(* POU GENERAL/FB_CALC_TOOLTENSION_FORCE_NEW, ST *)
FUNCTION_BLOCK FB_CALC_TOOLTENSION_FORCE_NEW
VAR_INPUT
	rForcePistonIn:REAL;	(* in Newton *)
	rPistonDiameterD1:REAL;	(* in mm *)
	rPistonDiameterD2:REAL;	(* in mm *)
	rMaxAirpressure:REAL;		(* in bar *)
	rFactorForce:REAL;
END_VAR
VAR_OUTPUT
	iAnalogOutput:INT;		(* range 0 - 32767 *)
	rSetMaxForce:REAL;		(* in Newton *)
	rForcePistonOut:REAL;	(* in Newton *)
END_VAR
VAR
	rMaxForce: REAL;
	rAreaOutside: REAL;
	rAreaInside: REAL;
	rArea: REAL;
	rTmpMaxAirpressure: REAL;
	rTmpAnalogOut:REAL;
END_VAR
(****************************************************************************************************************************************************)
(*****       This Functionblock calculate the effective value for the servo ventil for the ToolTension which the settled force         *****)
(****************************************************************************************************************************************************)
	rAreaOutside:=((rPistonDiameterD1/2)*(rPistonDiameterD1/2))*PI;
	rAreaInside:=((rPistonDiameterD2/2)*(rPistonDiameterD2/2))*PI;
	rArea:=ABS(rAreaOutside - rAreaInside);
	rArea:=rArea / 1000000.0;	(* Umwandeln von mm^2 in m^2 *)
	rTmpMaxAirpressure:=rMaxAirpressure * 100000.0;	(* convert from bar to pascal *)
	rMaxForce:=rArea * rTmpMaxAirpressure * rFactorForce;
	rSetMaxForce:=rMaxForce;

	IF(rMaxForce = 0) THEN rMaxForce:=0.01; END_IF;	(* check divide by zero *)
	IF(rMaxForce <> 0.0) THEN
		rTmpAnalogOut:=(rForcePistonIn/rMaxForce)*32767;	(* 32767 = 10V *)
		IF (rTmpAnalogOut > 32767) THEN
			iAnalogOutput:=32767;
		ELSE
			iAnalogOutput:=REAL_TO_INT(rTmpAnalogOut);
		END_IF;
		rForcePistonOut:=rForcePistonIn;
	ELSE
		iAnalogOutput:=0;
		rForcePistonOut:=0;
	END_IF;
END_FUNCTION_BLOCK

(* POU FB_HARDWARE/FBHW_CYL_STANDARD, ST *)
FUNCTION_BLOCK FBHW_CYL_STANDARD
VAR_INPUT
	xCtrlePosOn:BOOL;
	xCtrlePosOff:BOOL;
END_VAR
VAR_OUTPUT
	xCylinder:BOOL;
END_VAR
VAR_IN_OUT
	T_Cylinder:ST_CYLINDER;
END_VAR
VAR
(* variable *)
	xConfirmResetFB:BOOL:=FALSE;
	iStep:INT;
(* timer *)
	TimerOn:TON;
	TimerOff:TON;
	TimerPreOn:TON;
	TimerPreOff:TON;
	TimerOut:TON;
	TimerActiv: TON;
(* trigger *)
	RisingEdgeActiv:R_TRIG;
	FallingEdgeActiv:F_TRIG;
	RisingEdgeReset:R_TRIG;
	RisingEdgeExecute:R_TRIG;
	TimerAfterSensor: TON;
END_VAR
(* if function bloc set activ then Analog state will be transfered *)
	RisingEdgeActiv(CLK:=T_Cylinder.T_CtrleCyl.xFBActiv);
	FallingEdgeActiv(CLK:=T_Cylinder.T_CtrleCyl.xFBActiv);
	IF RisingEdgeActiv.Q OR FallingEdgeActiv.Q THEN
	(* set Analog Out = In on the rising edge from the activ signal *)
		xCylinder:=NOT(T_Cylinder.T_Config.xActivState);
		T_Cylinder.T_CtrleCyl.T_Standard.xActivOn:= FALSE;
	END_IF

(* if bloc disable if activ signal is inactiv *)
	IF T_Cylinder.T_CtrleCyl.xFBActiv THEN
	(* copy control position state *)
		T_Cylinder.T_CtrleCyl.xStatePosOn:=xCtrlePosOn;
		T_Cylinder.T_CtrleCyl.xStatePosOff:=xCtrlePosOff;
	ELSE
	(* exit FB *)
		T_Cylinder.T_CtrleCyl.xStatePosOn:=xCtrlePosOn;
		T_Cylinder.T_CtrleCyl.xStatePosOff:=xCtrlePosOff;
		RETURN;
	END_IF

(* wait for reseting *)
	RisingEdgeReset(CLK:=T_Cylinder.T_CtrleCyl.xReset);
	IF RisingEdgeReset.Q THEN
		(* Init. timer *)
		TimerOn(IN:=TRUE,PT:=T#1ms);
		TimerOff(IN:=TRUE,PT:=T#1ms);
		TimerPreOn(IN:=TRUE,PT:=T#1ms);
		TimerPreOff(IN:=TRUE,PT:=T#1ms);
		TimerOut(IN:=TRUE,PT:=T#1ms);
	(* Init. variable *)
		iStep:=0;
	(* Init. structure *)
		T_Cylinder.T_CtrleCyl.iFunction:=0;
		T_Cylinder.T_CtrleCyl.T_Standard.xActivOn:=FALSE;
		xCylinder:=NOT(T_Cylinder.T_Config.xActivState);
		T_Cylinder.T_CtrleCyl.xDone:=FALSE;
		T_Cylinder.T_CtrleCyl.xErr:=FALSE;
		T_Cylinder.T_CtrleCyl.udiErrorID:=16#0;
	(* confirm reset *)
		xConfirmResetFB:=TRUE;
	(* exit function *)
		RETURN;
	ELSE
		IF xConfirmResetFB THEN
		(* confirm reset FB *)
			T_Cylinder.T_CtrleCyl.xDone:=TRUE;
			T_Cylinder.T_CtrleCyl.xErr:=FALSE;
			T_Cylinder.T_CtrleCyl.udiErrorID:=16#0;
			(* reset variable *)
			xConfirmResetFB:=FALSE;
		END_IF
	END_IF

(* if bloc disable if activ signal is inactiv *)
	IF NOT(T_Cylinder.T_CtrleCyl.xFBActiv) THEN
		RETURN;
	END_IF

(* wait for execute *)
	RisingEdgeExecute(CLK:=T_Cylinder.T_CtrleCyl.xExecute);
	IF RisingEdgeExecute.Q THEN
		IF NOT(T_Cylinder.T_CtrleCyl.xDone) AND NOT(T_Cylinder.T_CtrleCyl.xErr) THEN
		(* can execute function if both signal are disable *)
			RETURN;
		END_IF
		CASE T_Cylinder.T_CtrleCyl.iFunction OF
		(* disable *)
		1:	iStep:=11;
		(* Activ without sensor position ctrle *)
		2:	iStep:=1;
		(* inverse cylinder state *)
		51:	iStep:=51;
		ELSE
			(* function not implemented *)
			iStep:=0;
			T_Cylinder.T_CtrleCyl.xDone:=FALSE;
			T_Cylinder.T_CtrleCyl.xErr:=TRUE;
			T_Cylinder.T_CtrleCyl.udiErrorID:=16#F000;
			(* exit FB *)
			RETURN;
		END_CASE
		(* Init. variable *)
		T_Cylinder.T_CtrleCyl.xDone:=FALSE;
		T_Cylinder.T_CtrleCyl.xErr:=FALSE;
		T_Cylinder.T_CtrleCyl.udiErrorID:=16#0;
		(* exit FB *)
		RETURN;
	END_IF

(* Timer activ *)
	TimerOn(IN:=TRUE,PT:=T_Cylinder.T_Config.tDelayOn);
	TimerOff(IN:=TRUE,PT:=T_Cylinder.T_Config.tDelayOff);
	TimerPreOn(IN:=TRUE,PT:=T_Cylinder.T_Config.tDelayPreOn);
	TimerPreOff(IN:=TRUE,PT:=T_Cylinder.T_Config.tDelayPreOff);
	TimerOut(IN:=TRUE,PT:=T_Cylinder.T_Config.tTimeOut);
	TimerActiv(IN:=TRUE,PT:=T_Cylinder.T_CtrleCyl.T_Standard.tDelayActiv);
	TimerAfterSensor(IN:=TRUE,PT:=T_Cylinder.T_CtrleCyl.T_Standard.tDelayAfterSensor);
(* waiting for activ *)
	CASE iStep OF
	(* process timer On *)
	1:	IF (T_Cylinder.T_Config.tDelayPreOn = T#0s) THEN
			TimerOn(IN:=FALSE);
			xCylinder:=T_Cylinder.T_Config.xActivState;
			T_Cylinder.T_CtrleCyl.T_Standard.xActivOn:=TRUE;
			iStep:=2;
		ELSE
			TimerPreOn(IN:=FALSE);
			iStep:=4;
		END_IF;
	(* wait for timer On *)
	2:	IF TimerOn.Q THEN
			iStep:=3;
			TimerOut(IN:=FALSE);
		END_IF
	(* control position activ *)
	3:	IF T_Cylinder.T_Config.xCtrlePosOn THEN
		(* position ctrle activ *)
			IF TimerOut.Q THEN
			(* timerout done, activ error cylinder has not activ position reached *)
				iStep:=999;
			ELSE
				IF xCtrlePosOn THEN
				(* Activ position reached, activ confirmation *)
					iStep:=80;
				END_IF
			END_IF
		ELSE
		(* no position ctrle, activ confirm *)
			iStep:=90;
		END_IF
	(* wait for timer Pre On *)
	4:	IF TimerPreOn.Q THEN
			T_Cylinder.T_Config.tDelayPreOn:=T#0s;
			iStep:=1;
		END_IF
	(* process timer Off *)
	11:	IF (T_Cylinder.T_Config.tDelayPreOff = T#0s) THEN
			TimerOff(IN:=FALSE);
			xCylinder:=NOT(T_Cylinder.T_Config.xActivState);
			T_Cylinder.T_CtrleCyl.T_Standard.xActivOn:=FALSE;
			iStep:=12;
		ELSE
			TimerPreOff(IN:=FALSE);
			iStep:=14;
		END_IF;
	(* wait for timer Off *)
	12:	IF TimerOff.Q THEN
			iStep:=13;
			TimerOut(IN:=FALSE);
		END_IF
	(* control position inactiv *)
	13:	IF T_Cylinder.T_Config.xCtrlePosOff THEN
		(* control position activ *)
			IF TimerOut.Q THEN
			(* timerout done, activ error 'cylinder has not inactiv position reached' *)
				iStep:=998;
			ELSE
				IF xCtrlePosOff THEN
				(* inactiv position reached, activ confirmation *)
					iStep:=85;
				END_IF
			END_IF
		ELSE
		(* no control position activ, activ confirmation *)
			iStep:=99;
		END_IF
	(* wait for timer Pre Off *)
	14:	IF TimerPreOff.Q THEN
			T_Cylinder.T_Config.tDelayPreOff:=T#0s;
			iStep:=11;
		END_IF
	(* inverse cylinder state *)
	51:	xCylinder:=NOT(xCylinder);
		T_Cylinder.T_CtrleCyl.T_Standard.xActivOn:=NOT(T_Cylinder.T_CtrleCyl.T_Standard.xActivOn);
		iStep:=99;
	80:	IF (T_Cylinder.T_CtrleCyl.T_Standard.tDelayAfterSensor <> T#0s) THEN
			TimerAfterSensor(IN:=FALSE);
			iStep:=81;
		ELSE
			iStep:=90;
		END_IF;
	(* wait for time after sensor *)
	81:	IF TimerAfterSensor.Q THEN
			iStep:=90;
		END_IF
	85:	IF (T_Cylinder.T_CtrleCyl.T_Standard.tDelayAfterSensor <> T#0s) THEN
			TimerAfterSensor(IN:=FALSE);
			iStep:=86;
		ELSE
			iStep:=99;
		END_IF;
	(* wait for time after sensor *)
	86:	IF TimerAfterSensor.Q THEN
			iStep:=99;
		END_IF
	(* test if delay activ *)
	90:	IF T_Cylinder.T_CtrleCyl.T_Standard.tDelayActiv <> T#0s THEN
			TimerActiv(IN:=FALSE);
			iStep:=98;
		ELSE
			iStep:=99;
		END_IF
	(* wait for time delay activ *)
	98:	IF TimerActiv.Q THEN
		(* activ time is over, set variable off *)
			xCylinder:=NOT(T_Cylinder.T_Config.xActivState);
			T_Cylinder.T_CtrleCyl.T_Standard.xActivOn:=FALSE;
			iStep:=99;
		END_IF
	(* process end *)
	99:	T_Cylinder.T_CtrleCyl.xDone:=TRUE;
		T_Cylinder.T_CtrleCyl.xErr:=FALSE;
		T_Cylinder.T_CtrleCyl.udiErrorID:=16#0;
	(* error, cylinder not in inactiv position *)
	998:	T_Cylinder.T_CtrleCyl.xDone:=FALSE;
		T_Cylinder.T_CtrleCyl.xErr:=TRUE;
		T_Cylinder.T_CtrleCyl.udiErrorID:=16#F202;
	(* error, cylinder not in activ position *)
	999:	T_Cylinder.T_CtrleCyl.xDone:=FALSE;
		T_Cylinder.T_CtrleCyl.xErr:=TRUE;
		T_Cylinder.T_CtrleCyl.udiErrorID:=16#F201;
	END_CASE
END_FUNCTION_BLOCK

(* POU PRG_TWINSAFE, FBD *)
PROGRAM PRG_TWINSAFE
VAR
	TwinSAFEinputKlemme1: TwinSAFE_input;
	TwinSAFEinputKlemme2: TwinSAFE_input;
	TwinSAFEinputKlemme3: TwinSAFE_input;
END_VAR
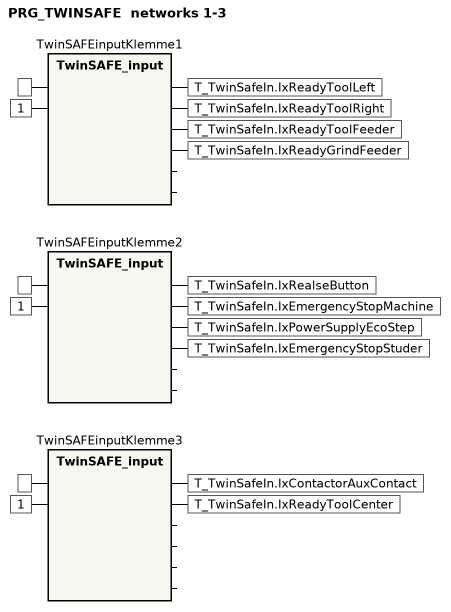
_FBD_ (* Function Block Diagram *)
NETWORK 1 (* Read of the TwinSAFE inputs *)
	TwinSAFEinputKlemme1:TwinSAFE_input(, 1, out 2 => T_TwinSafeIn.IxReadyToolRight, out 3 => T_TwinSafeIn.IxReadyToolFeeder, out 4 => T_TwinSafeIn.IxReadyGrindFeeder) => T_TwinSafeIn.IxReadyToolLeft
NETWORK 2 (* Read of the TwinSAFE inputs *)
	TwinSAFEinputKlemme2:TwinSAFE_input(, 1, out 2 => T_TwinSafeIn.IxEmergencyStopMachine, out 3 => T_TwinSafeIn.IxPowerSupplyEcoStep, out 4 => T_TwinSafeIn.IxEmergencyStopStuder) => T_TwinSafeIn.IxRealseButton
NETWORK 3 (* Read of the TwinSAFE inputs *)
	TwinSAFEinputKlemme3:TwinSAFE_input(, 1, out 2 => T_TwinSafeIn.IxReadyToolCenter) => T_TwinSafeIn.IxContactorAuxContact
_END_FBD_
END_PROGRAM

(* POU PRG_USB_IO_PANEL, ST *)
PROGRAM PRG_USB_IO_PANEL
VAR
(* Panel tastatur *)
	(* function bloc *)
	fbCtrlePanel_IO:FBHW_PANEL_IO;
	(* IO connection *)

	IarxCtrlePanelButton AT %I* : ARRAY[1..10] OF BOOL;
	QarxCtrlePanelLed AT %Q* : ARRAY[1..10] OF BOOL;
END_VAR
(****************************************************************************************************************************************************)
(***********                This Programm Unit make the connection for read and set the ControlPanel Led and Button               ************)
(****************************************************************************************************************************************************)
(* Call FB *)
	fbCtrlePanel_IO(	arxButton:=IarxCtrlePanelButton,
					T_CtrlePanel:=T_CtrlePanel,
					arxLed=>QarxCtrlePanelLed);
END_PROGRAM

(* POU FB_HARDWARE/FBHW_PANEL_IO, ST *)
FUNCTION_BLOCK FBHW_PANEL_IO
VAR_INPUT
	arxButton:ARRAY[1..10] OF BOOL;
END_VAR
VAR_OUTPUT
	arxLed:ARRAY[1..10] OF BOOL;
END_VAR
VAR_IN_OUT
	T_CtrlePanel:ST_CTRLEPANEL;
END_VAR
VAR
(* variable *)
	xConfirmResetFB:BOOL;
	xConfirmFct:BOOL;
	i: INT;
	si: SINT;
(* trigger *)
	RisingEdgeExecute:R_TRIG;
	RisingEdgeReset:R_TRIG;
END_VAR
(****************************************************************************************************************************************************)
(***********                                            This Functionblock is for manage the IO's of the ControlPanel                                             ************)
(****************************************************************************************************************************************************)
(* reset function bloc *)
	RisingEdgeReset(CLK:=T_CtrlePanel.xReset);
	IF RisingEdgeReset.Q THEN
	(* reset output *)
		FOR i := 1 TO 10 DO
			arxLed[i]:=FALSE;
		END_FOR
	(* init. structure *)
		T_CtrlePanel.iFunction:=0;
		T_CtrlePanel.xDone:=FALSE;
		T_CtrlePanel.xErr:=FALSE;
		T_CtrlePanel.udiErrorID:=0;
		T_CtrlePanel.udiButton:=0;
		T_CtrlePanel.udiLED:=0;
	(* confirm reset *)
		xConfirmResetFB:=TRUE;
	(* exit fb *)
		RETURN;
	ELSE
		IF xConfirmResetFB THEN
		(* confirm reset FB *)
			T_CtrlePanel.xDone:=TRUE;
			T_CtrlePanel.xErr:=FALSE;
			T_CtrlePanel.udiErrorID:=0;
			(* Init. variable *)
			xConfirmResetFB:=FALSE;
		END_IF
	END_IF

(* Switch on/off the Led from the control panel *)
	RisingEdgeExecute(CLK:=T_CtrlePanel.xExecute);
	IF RisingEdgeExecute.Q THEN
		CASE T_CtrlePanel.iFunction OF
		(* switch off a specific LED off *)
		-10..-1:	IF arxLed[ABS(T_CtrlePanel.iFunction)] THEN
					arxLed[ABS(T_CtrlePanel.iFunction)]:=FALSE;
					T_CtrlePanel.udiLED:=T_CtrlePanel.udiLED - MUX(ABS(T_CtrlePanel.iFunction)-1,1,2,4,8,16,32,64,128,256,512);
				END_IF
		(* switch off all the LED *)
		0:	FOR i := 1 TO 10 DO
				arxLed[i]:=FALSE;
			END_FOR
			T_CtrlePanel.udiLED:=0;
		(* switch on a specific Led on *)
		1..10:	IF NOT(arxLed[T_CtrlePanel.iFunction]) THEN
					arxLed[T_CtrlePanel.iFunction]:=TRUE;
					T_CtrlePanel.udiLED:=T_CtrlePanel.udiLED + MUX(T_CtrlePanel.iFunction-1,1,2,4,8,16,32,64,128,256,512);
				END_IF
		ELSE
			(* function not implemented *)
			T_CtrlePanel.xDone:=FALSE;
			T_CtrlePanel.xErr:=TRUE;
			T_CtrlePanel.udiErrorID:=16#F000;
			(* exit FB *)
			RETURN;
		END_CASE
		(* Init. variable *)
		T_CtrlePanel.xDone:=FALSE;
		T_CtrlePanel.xErr:=FALSE;
		T_CtrlePanel.udiErrorID:=16#0;
		(* activ confirm *)
		xConfirmFct:=TRUE;
		(* exit FB *)
		RETURN;
	END_IF

(* return the button state *)
	T_CtrlePanel.udiButton:=0;
	FOR i := 0 TO 9 DO
		IF arxButton[i+1] THEN
			T_CtrlePanel.udiButton:=T_CtrlePanel.udiButton + MUX(i,1,2,4,8,16,32,64,128,256,512);
		END_IF
	END_FOR

(* set the led state *)
	FOR si := 0 TO 9 DO
		IF GETBIT32(T_CtrlePanel.udiLED,si) <> 16#0 THEN
			arxLed[si+1]:=TRUE; ELSE arxLed[si+1]:=FALSE; END_IF
	END_FOR

(* wait to confirm *)
	IF xConfirmFct THEN
		T_CtrlePanel.xDone:=TRUE;
		T_CtrlePanel.xErr:=FALSE;
		T_CtrlePanel.udiErrorID:=16#0;
		(* reset variable *)
		xConfirmFct:=FALSE;
	END_IF
END_FUNCTION_BLOCK

(* POU GENERAL/FB_CALC_TOOLTENSION_FORCE, ST *)
FUNCTION_BLOCK FB_CALC_TOOLTENSION_FORCE
VAR_INPUT
	rForcePistonIn:REAL;	(* in Newton *)
	rPistonDiameterD:REAL;	(* in mm *)
	rMaxAirpressure:REAL;		(* in bar *)
END_VAR
VAR_OUTPUT
	iAnalogOutput:INT;		(* range 0 - 32767 *)
	rSetMaxForce:REAL;		(* in Newton *)
	rForcePistonOut:REAL;		(* in Newton *)
END_VAR
VAR
	rMaxForce: REAL;
	rAreaOutside: REAL;
	rArea: REAL;
	rTmpMaxAirpressure: REAL;
	rTmpAnalogOut:REAL;
END_VAR
(****************************************************************************************************************************************************)
(*****       This Functionblock calculate the effective value for the servo ventil for the ToolTension which the settled force         *****)
(****************************************************************************************************************************************************)
	rAreaOutside:=((rPistonDiameterD/2)*(rPistonDiameterD/2))*PI;
	rArea:=rAreaOutside;
	rArea:=rArea / 1000000.0;	(* calculate from mm^2 to m^2 *)
	rTmpMaxAirpressure:=rMaxAirpressure * 100000.0;	(* convert from bar to pascal *)
	rMaxForce:=rArea * rTmpMaxAirpressure;
	rSetMaxForce:=rMaxForce;
	IF(rMaxForce = 0) THEN rMaxForce:=0.01; END_IF;	(* check divide by zero *)
	IF(rMaxForce <> 0.0) THEN
		rTmpAnalogOut:=(rForcePistonIn/rMaxForce)*32767;	(* 32767 = 10V *)
		IF (rTmpAnalogOut > 32767) THEN
			iAnalogOutput:=32767;
		ELSE
			iAnalogOutput:=REAL_TO_INT(rTmpAnalogOut);
		END_IF;
		rForcePistonOut:=rForcePistonIn;
	ELSE
		iAnalogOutput:=0;
		rForcePistonOut:=0;
	END_IF;
END_FUNCTION_BLOCK
